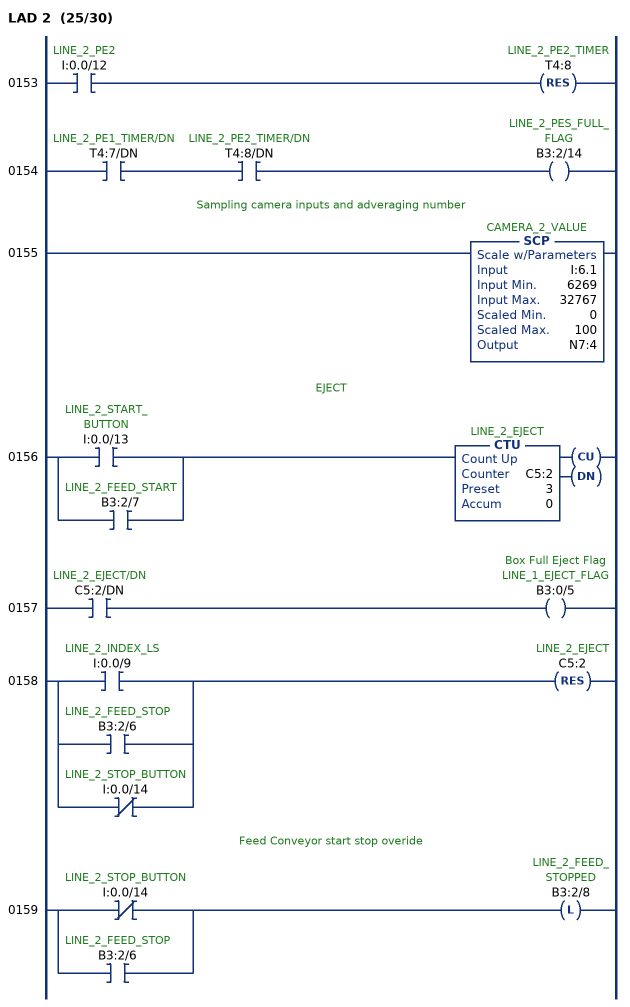
% Rung: 153 %  % edit flag set %
SOR XIC I:0.0/12 RES T4:8 EOR
%   I:0.0/12  LINE_2_PE2 %
%   T4:8  LINE_2_PE2_TIMER %
% Rung: 154 %  % edit flag set %
SOR XIC T4:7/DN XIC T4:8/DN OTE B3:2/14 EOR
%   T4:7  LINE_2_PE1_TIMER %
%   T4:8  LINE_2_PE2_TIMER %
%   B3:2/14  LINE_2_PES_FULL_FLAG %
% Rung: 155 %  % edit flag set %
% Sampling camera inputs and adveraging number %
SOR SCP I:6.1 6269 32767 0 100 N7:4 EOR
%   N7:4  CAMERA_2_VALUE %
% Rung: 156 %  % edit flag set %
% EJECT %
SOR BST XIC I:0.0/13 NXB XIC B3:2/7 BND CTU C5:2 3 0 EOR
%   I:0.0/13  LINE_2_START_BUTTON %
%   B3:2/7  LINE_2_FEED_START %
%   C5:2  LINE_2_EJECT %
% Rung: 157 %  % edit flag set %
SOR XIC C5:2/DN OTE B3:0/5 EOR
%   C5:2  LINE_2_EJECT %
%   B3:0/5  LINE_1_EJECT_FLAG  "Box Full Eject Flag" %
% Rung: 158 %  % edit flag set %
SOR BST XIC I:0.0/9 NXB BST XIC B3:2/6 NXB XIO I:0.0/14 BND BND RES C5:2 EOR
%   I:0.0/9  LINE_2_INDEX_LS %
%   B3:2/6  LINE_2_FEED_STOP %
%   I:0.0/14  LINE_2_STOP_BUTTON %
%   C5:2  LINE_2_EJECT %
% Rung: 159 %  % edit flag set %
% Feed Conveyor start stop overide %
SOR BST XIO I:0.0/14 NXB XIC B3:2/6 BND OTL B3:2/8 EOR
%   I:0.0/14  LINE_2_STOP_BUTTON %
%   B3:2/6  LINE_2_FEED_STOP %
%   B3:2/8  LINE_2_FEED_STOPPED %

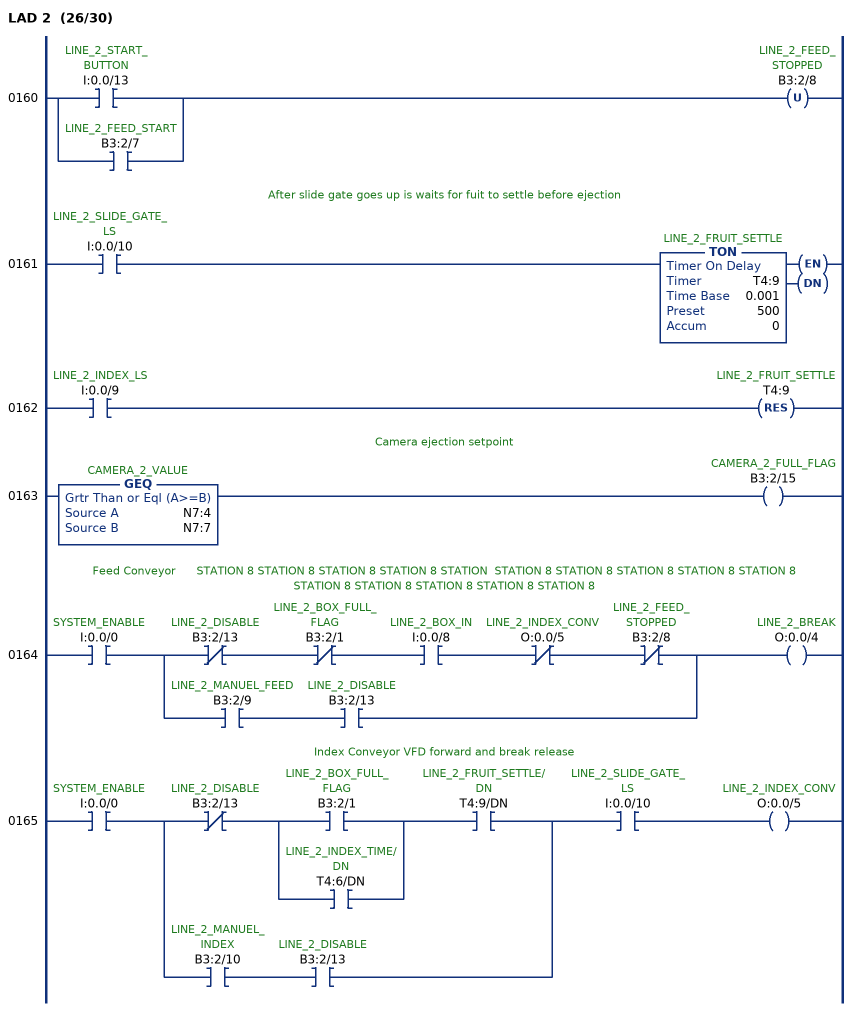
% Rung: 160 %  % edit flag set %
SOR BST XIC I:0.0/13 NXB XIC B3:2/7 BND OTU B3:2/8 EOR
%   I:0.0/13  LINE_2_START_BUTTON %
%   B3:2/7  LINE_2_FEED_START %
%   B3:2/8  LINE_2_FEED_STOPPED %
% Rung: 161 %  % edit flag set %
% After slide gate goes up is waits for fuit to settle before ejection %
SOR XIC I:0.0/10 TON T4:9 0.001 500 0 EOR
%   I:0.0/10  LINE_2_SLIDE_GATE_LS %
%   T4:9  LINE_2_FRUIT_SETTLE %
% Rung: 162 %  % edit flag set %
SOR XIC I:0.0/9 RES T4:9 EOR
%   I:0.0/9  LINE_2_INDEX_LS %
%   T4:9  LINE_2_FRUIT_SETTLE %
% Rung: 163 %  % edit flag set %
% Camera ejection setpoint %
SOR GEQ N7:4 N7:7 OTE B3:2/15 EOR
%   N7:4  CAMERA_2_VALUE %
%   N7:7  LINE_2_CAMERA_EJECT %
%   B3:2/15  CAMERA_2_FULL_FLAG %
% Rung: 164 %  % edit flag set %
% Feed Conveyor      STATION 8 STATION 8 STATION 8 STATION 8 STATION  STATION 8 STATION 8 STATION 8 STATION 8 STATION 8 STATION 8 STATION 8 STATION 8 STATION 8 STATION 8 %
SOR XIC I:0.0/0 BST XIO B3:2/13 XIO B3:2/1 XIC I:0.0/8 XIO O:0.0/5 XIO B3:2/8 NXB XIC B3:2/9 XIC B3:2/13 BND OTE O:0.0/4 EOR
%   I:0.0/0  SYSTEM_ENABLE %
%   B3:2/13  LINE_2_DISABLE %
%   B3:2/1  LINE_2_BOX_FULL_FLAG %
%   I:0.0/8  LINE_2_BOX_IN %
%   O:0.0/5  LINE_2_INDEX_CONV %
%   B3:2/8  LINE_2_FEED_STOPPED %
%   B3:2/9  LINE_2_MANUEL_FEED %
%   O:0.0/4  LINE_2_BREAK %
% Rung: 165 %  % edit flag set %
% Index Conveyor VFD forward and break release %
SOR XIC I:0.0/0 BST XIO B3:2/13 BST XIC B3:2/1 NXB XIC T4:6/DN BND XIC T4:9/DN NXB XIC B3:2/10 XIC B3:2/13 BND XIC I:0.0/10 OTE O:0.0/5 EOR
%   I:0.0/0  SYSTEM_ENABLE %
%   B3:2/13  LINE_2_DISABLE %
%   B3:2/1  LINE_2_BOX_FULL_FLAG %
%   T4:6  LINE_2_INDEX_TIME %
%   T4:9  LINE_2_FRUIT_SETTLE %
%   B3:2/10  LINE_2_MANUEL_INDEX %
%   I:0.0/10  LINE_2_SLIDE_GATE_LS %
%   O:0.0/5  LINE_2_INDEX_CONV %

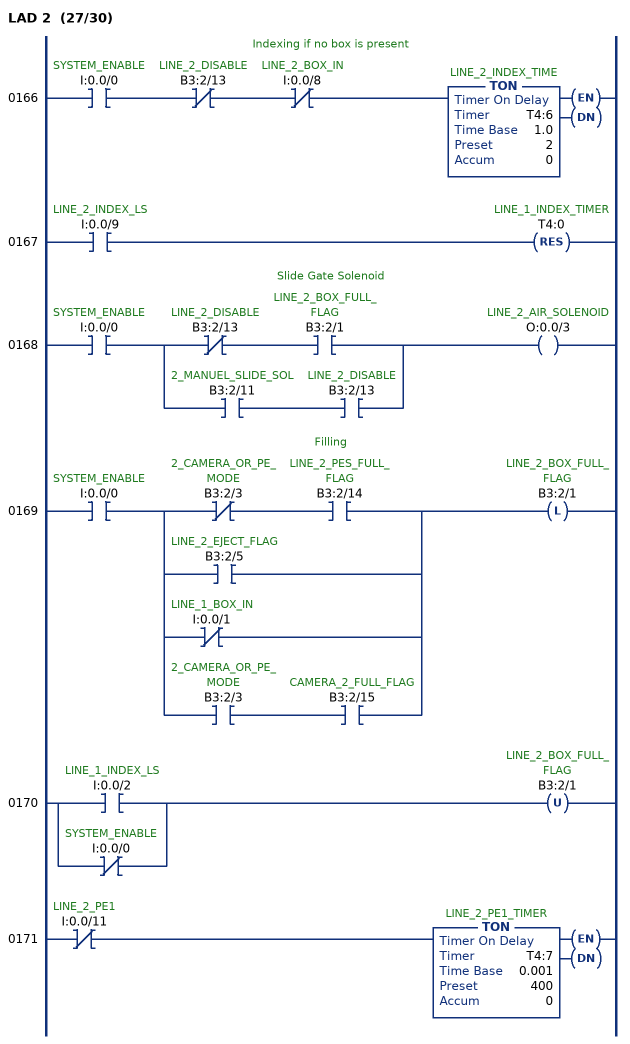
% Rung: 166 %  % edit flag set %
% Indexing if no box is present %
SOR XIC I:0.0/0 XIO B3:2/13 XIO I:0.0/8 TON T4:6 1.0 2 0 EOR
%   I:0.0/0  SYSTEM_ENABLE %
%   B3:2/13  LINE_2_DISABLE %
%   I:0.0/8  LINE_2_BOX_IN %
%   T4:6  LINE_2_INDEX_TIME %
% Rung: 167 %  % edit flag set %
SOR XIC I:0.0/9 RES T4:0 EOR
%   I:0.0/9  LINE_2_INDEX_LS %
%   T4:0  LINE_1_INDEX_TIMER %
% Rung: 168 %  % edit flag set %
% Slide Gate Solenoid %
SOR XIC I:0.0/0 BST XIO B3:2/13 XIC B3:2/1 NXB XIC B3:2/11 XIC B3:2/13 BND OTE O:0.0/3 EOR
%   I:0.0/0  SYSTEM_ENABLE %
%   B3:2/13  LINE_2_DISABLE %
%   B3:2/1  LINE_2_BOX_FULL_FLAG %
%   B3:2/11  2_MANUEL_SLIDE_SOL %
%   O:0.0/3  LINE_2_AIR_SOLENOID %
% Rung: 169 %  % edit flag set %
% Filling %
SOR XIC I:0.0/0 BST XIO B3:2/3 XIC B3:2/14 NXB BST XIC B3:2/5 NXB BST XIO I:0.0/1 NXB XIC B3:2/3 XIC B3:2/15 BND BND BND OTL B3:2/1 EOR
%   I:0.0/0  SYSTEM_ENABLE %
%   B3:2/3  2_CAMERA_OR_PE_MODE %
%   B3:2/14  LINE_2_PES_FULL_FLAG %
%   B3:2/5  LINE_2_EJECT_FLAG %
%   I:0.0/1  LINE_1_BOX_IN %
%   B3:2/15  CAMERA_2_FULL_FLAG %
%   B3:2/1  LINE_2_BOX_FULL_FLAG %
% Rung: 170 %  % edit flag set %
SOR BST XIC I:0.0/2 NXB XIO I:0.0/0 BND OTU B3:2/1 EOR
%   I:0.0/2  LINE_1_INDEX_LS %
%   I:0.0/0  SYSTEM_ENABLE %
%   B3:2/1  LINE_2_BOX_FULL_FLAG %
% Rung: 171 %  % edit flag set %
SOR XIO I:0.0/11 TON T4:7 0.001 400 0 EOR
%   I:0.0/11  LINE_2_PE1 %
%   T4:7  LINE_2_PE1_TIMER %

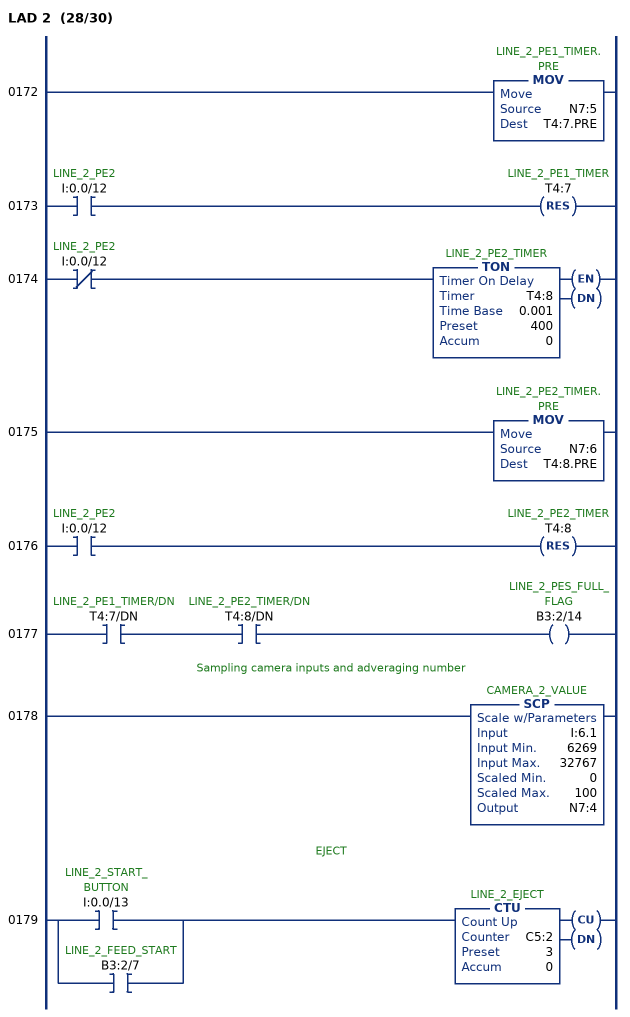
% Rung: 172 %  % edit flag set %
SOR MOV N7:5 T4:7.PRE EOR
%   N7:5  LINE_2_PE1_TIME_MOV %
%   T4:7  LINE_2_PE1_TIMER %
% Rung: 173 %  % edit flag set %
SOR XIC I:0.0/12 RES T4:7 EOR
%   I:0.0/12  LINE_2_PE2 %
%   T4:7  LINE_2_PE1_TIMER %
% Rung: 174 %  % edit flag set %
SOR XIO I:0.0/12 TON T4:8 0.001 400 0 EOR
%   I:0.0/12  LINE_2_PE2 %
%   T4:8  LINE_2_PE2_TIMER %
% Rung: 175 %  % edit flag set %
SOR MOV N7:6 T4:8.PRE EOR
%   N7:6  LINE_2_PE2_TIME_MOV %
%   T4:8  LINE_2_PE2_TIMER %
% Rung: 176 %  % edit flag set %
SOR XIC I:0.0/12 RES T4:8 EOR
%   I:0.0/12  LINE_2_PE2 %
%   T4:8  LINE_2_PE2_TIMER %
% Rung: 177 %  % edit flag set %
SOR XIC T4:7/DN XIC T4:8/DN OTE B3:2/14 EOR
%   T4:7  LINE_2_PE1_TIMER %
%   T4:8  LINE_2_PE2_TIMER %
%   B3:2/14  LINE_2_PES_FULL_FLAG %
% Rung: 178 %  % edit flag set %
% Sampling camera inputs and adveraging number %
SOR SCP I:6.1 6269 32767 0 100 N7:4 EOR
%   N7:4  CAMERA_2_VALUE %
% Rung: 179 %  % edit flag set %
% EJECT %
SOR BST XIC I:0.0/13 NXB XIC B3:2/7 BND CTU C5:2 3 0 EOR
%   I:0.0/13  LINE_2_START_BUTTON %
%   B3:2/7  LINE_2_FEED_START %
%   C5:2  LINE_2_EJECT %

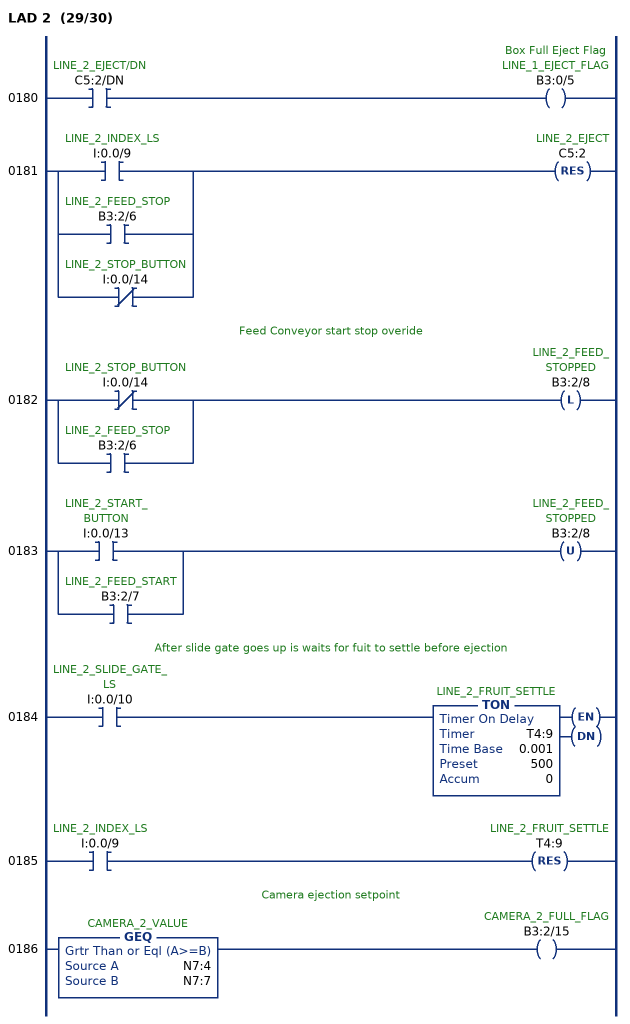
% Rung: 180 %  % edit flag set %
SOR XIC C5:2/DN OTE B3:0/5 EOR
%   C5:2  LINE_2_EJECT %
%   B3:0/5  LINE_1_EJECT_FLAG  "Box Full Eject Flag" %
% Rung: 181 %  % edit flag set %
SOR BST XIC I:0.0/9 NXB BST XIC B3:2/6 NXB XIO I:0.0/14 BND BND RES C5:2 EOR
%   I:0.0/9  LINE_2_INDEX_LS %
%   B3:2/6  LINE_2_FEED_STOP %
%   I:0.0/14  LINE_2_STOP_BUTTON %
%   C5:2  LINE_2_EJECT %
% Rung: 182 %  % edit flag set %
% Feed Conveyor start stop overide %
SOR BST XIO I:0.0/14 NXB XIC B3:2/6 BND OTL B3:2/8 EOR
%   I:0.0/14  LINE_2_STOP_BUTTON %
%   B3:2/6  LINE_2_FEED_STOP %
%   B3:2/8  LINE_2_FEED_STOPPED %
% Rung: 183 %  % edit flag set %
SOR BST XIC I:0.0/13 NXB XIC B3:2/7 BND OTU B3:2/8 EOR
%   I:0.0/13  LINE_2_START_BUTTON %
%   B3:2/7  LINE_2_FEED_START %
%   B3:2/8  LINE_2_FEED_STOPPED %
% Rung: 184 %  % edit flag set %
% After slide gate goes up is waits for fuit to settle before ejection %
SOR XIC I:0.0/10 TON T4:9 0.001 500 0 EOR
%   I:0.0/10  LINE_2_SLIDE_GATE_LS %
%   T4:9  LINE_2_FRUIT_SETTLE %
% Rung: 185 %  % edit flag set %
SOR XIC I:0.0/9 RES T4:9 EOR
%   I:0.0/9  LINE_2_INDEX_LS %
%   T4:9  LINE_2_FRUIT_SETTLE %
% Rung: 186 %  % edit flag set %
% Camera ejection setpoint %
SOR GEQ N7:4 N7:7 OTE B3:2/15 EOR
%   N7:4  CAMERA_2_VALUE %
%   N7:7  LINE_2_CAMERA_EJECT %
%   B3:2/15  CAMERA_2_FULL_FLAG %

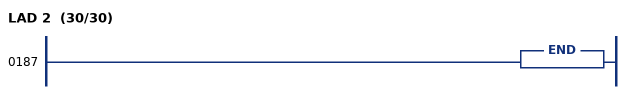
% Rung: 187 %
SOR END EOR

OTHER DOCUMENTED ADDRESSES
  B3:0/4  1_BOX_FULL_UNLATCH  "Box Full Unlatch"
  B3:2/4  2_BOX_FULL_UNLATCH
  B3:3/4  3_BOX_FULL_UNLATCH
  B3:4/4  4_BOX_FULL_UNLATCH
  B3:5/4  5_BOX_FULL_UNLATCH
  B3:6/1  LINE_6_BOX_FULL_FLAG
  B3:6/3  6_CAMERA_OR_PE_MODE
  B3:6/4  6_BOX_FULL_UNLATCH
  B3:6/5  LINE_6_EJECT_FLAG
  B3:6/6  LINE_6_FEED_STOP
  B3:6/7  LINE_6_FEED_START
  B3:6/8  LINE_6_FEED_STOPPED
  B3:6/9  LINE_6_MANUAL_FEED
  B3:6/10  LINE_6_MANUAL_INDEX
  B3:6/11  6_MANUAL_SLIDE_SOL
  B3:6/13  LINE_6_DISABLE
  B3:6/14  LINE_6_PES_FULL_FLAG
  B3:6/15  CAMERA_6_FULL_FLAG
  B3:7/1  LINE_7_BOX_FULL_FLAG
  B3:7/3  7_CAMERA_OR_PE_MODE
  B3:7/4  7_BOX_FULL_UNLATCH
  B3:7/5  LINE_7_EJECT_FLAG
  B3:7/6  LINE_7_FEED_STOP
  B3:7/7  LINE_7_FEED_START
  B3:7/8  LINE_7_FEED_STOPPED
  B3:7/9  LINE_7_MANUAL_FEED
  B3:7/10  LINE_7_MANUAL_INDEX
  B3:7/11  7_MANUAL_SLIDE_SOL
  B3:7/13  LINE_7_DISABE
  B3:7/14  LINE_7_PES_FULL_FLAG
  B3:7/15  CAMERA_7_FULL_FLAG
  B3:8/3  8_CAMERA_OR_PE_MODE
  B3:8/4  8_BOX_FULL_UNLATCH
  B3:8/5  LINE_8_EJECT_FLAG
  B3:8/6  LINE_8_FEED_STOP
  B3:8/7  LINE_8_FEED_START
  B3:8/8  LINE_8_FEED_STOPPED
  B3:8/9  LINE_8_MANUAL_FEED
  B3:8/10  LINE_8_MANUAL_INDEX
  B3:8/11  8_MANUAL_SLIDE_SOL
  B3:8/13  LINE_8_DISABLE
  B3:8/14  LINE_8_PES_FULL_FLAG
  B3:8/15  CAMERA_8_FULL_FLAG
  C5:0.ACC  "Counter"
  C5:0/DN  COUNT_DONE
  C5:6  LINE_6_EJECT
  C5:7  LINE_7_EJECT
  I:2.0/0  LINE_6_BOX_IN
  I:2.0/1  LINE_6_INDEX_LS
  I:2.0/2  LINE_6_SLIDE_GATE_LS
  I:2.0/3  LINE_6_PE1
  I:2.0/4  LINE_6_PE2
  I:2.0/5  LINE_6_START_BUTTON
  I:2.0/6  LINE_6_STOP_BUTTON
  I:2.0/7  LINE_7_BOX_IN
  I:2.0/8  LINE_7_INDEX_LS
  I:2.0/9  LINE_7_SLIDE_GATE_LS
  I:2.0/10  LINE_7_PE1
  I:2.0/11  LINE_7_PE2
  I:2.0/12  LINE_7_START_BUTTON
  I:2.0/13  LINE_7_STOP_BUTTON
  I:2.0/14  LINE_8_BOX_IN
  I:2.0/15  LINE_8_INDEX_LS
  I:3.0/0  LINE_8_SLIDE_GATE_LS
  I:3.0/1  LINE_8_PE1
  I:3.0/2  LINE_8_PE2
  I:3.0/3  LINE_8_START_BUTTON
  I:3.0/4  LINE_8_STOP_BUTTON
  I:6.0/0  CAMERA_1  "Camera 1 4-20 input"
  I:7.0/0  CAMERA_5  "Camera 1 4-20 input"
  N7:20  CAMERA_6_VALUE
  N7:21  LINE_6_PE1_TIME_MOV
  N7:22  LINE_6_PE2_TIME_MOV
  N7:23  CAMERA_6_EJECT
  N7:24  CAMERA_7_VALUE
  N7:25  LINE_7_PE1_TIME_MOV
  N7:26  LINE_7_PE2_TIME_MOV
  N7:27  CAMERA_7_EJECT
  N7:28  CAMERA_8_VALUE
  N7:29  LINE_8_PE1_TIME_MOV
  N7:30  LINE_8_PE2_TIME_MOV
  N7:31  CAMERA_8_EJECT
  O:4.0/3  LINE_6_AIR_SOLENOID
  O:4.0/4  LINE_6_BREAK
  O:4.0/5  LINE_6_INDEX_CONV
  O:4.0/6  LINE_7_AIR_SOLENOID
  O:4.0/7  LINE_7_BREAK
  O:4.0/8  LINE_7_INDEX_CONV
  T4:22  LINE_6_INDEX_TIMER
  T4:23  LINE_6_PE1_TIMER
  T4:24  LINE_6_PE2_TIMER
  T4:25  LINE_6_FRUIT_SETTLE
  T4:26  LINE_7_INDEX_TIMER
  T4:27  LINE_7_PE1_TIMER
  T4:28  LINE_7_PE2_TIMER
  T4:29  LINE_7_FRUIT_SETTLE
  T4:30  LINE_8_INDEX_TIMER
  T4:31  LINE_8_PE1_TIMER
  T4:32  LINE_8_PE2_TIMER
  T4:33  LINE_8_FRUIT_SETTLE

REVISION NOTES
  0: Simplified

DATA TABLE (non-zero values as saved)
DATA B3
% B3:0 % 0X0004 0X000B 0X0000 0X0000 0X0000 0X0000 0X0000 0X0000 0X0000 0X0001
DATA T4
% .PRE .ACC %
% T4:0 % 2 0
% T4:1 % 400 0
% T4:2 % 1 1
% T4:3 % 1 0
% T4:4 % 400 0
% T4:5 % 500 0
% T4:6 % 1440 1530
DATA C5
% .PRE .ACC %
% C5:0 % 6 1
% C5:1 % 3 0
DATA N7
% N7:0 % 36 51 51 51 51 52 102 153 204 256
% N7:10 % 51 1470 400 400 50 0 0 0 0 0
DATA F8
% F8:0 % 0 22161 86.55965
